Fanuc TP program (LS listing): S005.LS

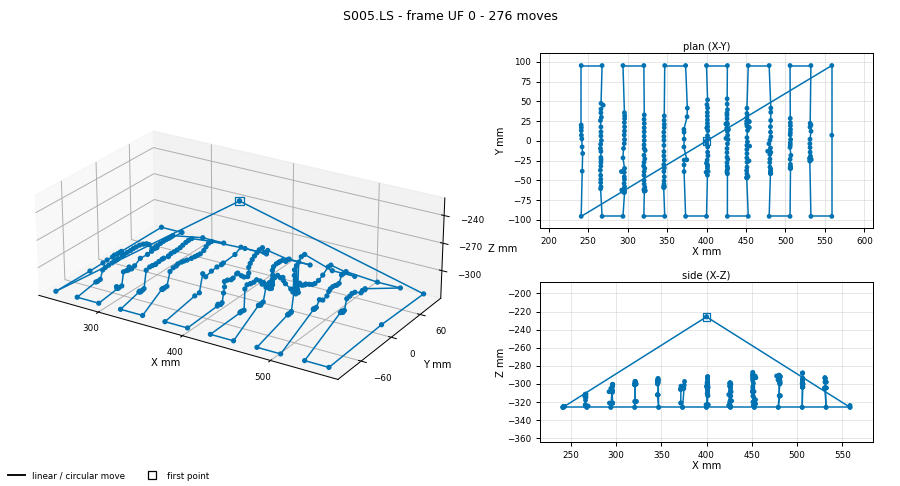
[picture p0: tool path of S005.LS in frame UF 0, 276 of 276 moves have a stored position in this frame; points joined in program order, loops and branches not executed]
/PROG  S005.LS
/ATTR
OWNER       = MNEDITOR;
COMMENT     = "";
PROG_SIZE   = 636;
CREATE      = DATE 23-01-07  TIME 11:59:14;
MODIFIED    = DATE 23-01-07  TIME 12:02:18;
FILE_NAME   = ;
VERSION     = 0;
LINE_COUNT  = 4;
MEMORY_SIZE = 992;
PROTECT     = READ_WRITE;
TCD:  STACK_SIZE    = 0,
      TASK_PRIORITY = 50,
      TIME_SLICE    = 0,
      BUSY_LAMP_OFF = 0,
      ABORT_REQUEST = 0,
      PAUSE_REQUEST = 0;
DEFAULT_GROUP    = 1,*,*,*,*;
CONTROL_CODE     = 00000000 00000000;
/MN
   1:J P[1] 100% FINE    ;
   2:L P[2] 300mm/sec CNT100    ;
   3:L P[3] 300mm/sec CNT100    ;
   4:L P[4] 300mm/sec CNT100    ;
   5:L P[5] 300mm/sec CNT100    ;
   6:L P[6] 300mm/sec CNT100    ;
   7:L P[7] 300mm/sec CNT100    ;
   8:L P[8] 300mm/sec CNT100    ;
   9:L P[9] 300mm/sec CNT100    ;
   10:L P[10] 300mm/sec CNT100    ;
   11:L P[11] 300mm/sec CNT100    ;
   12:L P[12] 300mm/sec CNT100    ;
   13:L P[13] 300mm/sec CNT100    ;
   14:L P[14] 300mm/sec CNT100    ;
   15:L P[15] 300mm/sec CNT100    ;
   16:L P[16] 300mm/sec CNT100    ;
   17:L P[17] 300mm/sec CNT100    ;
   18:L P[18] 300mm/sec CNT100    ;
   19:L P[19] 300mm/sec CNT100    ;
   20:L P[20] 300mm/sec CNT100    ;
   21:L P[21] 300mm/sec CNT100    ;
   22:L P[22] 300mm/sec CNT100    ;
   23:L P[23] 300mm/sec CNT100    ;
   24:L P[24] 300mm/sec CNT100    ;
   25:L P[25] 300mm/sec CNT100    ;
   26:L P[26] 300mm/sec CNT100    ;
   27:L P[27] 300mm/sec CNT100    ;
   28:L P[28] 300mm/sec CNT100    ;
   29:L P[29] 300mm/sec CNT100    ;
   30:L P[30] 300mm/sec CNT100    ;
   31:L P[31] 300mm/sec CNT100    ;
   32:L P[32] 300mm/sec CNT100    ;
   33:L P[33] 300mm/sec CNT100    ;
   34:L P[34] 300mm/sec CNT100    ;
   35:L P[35] 300mm/sec CNT100    ;
   36:L P[36] 300mm/sec CNT100    ;
   37:L P[37] 300mm/sec CNT100    ;
   38:L P[38] 300mm/sec CNT100    ;
   39:L P[39] 300mm/sec CNT100    ;
   40:L P[40] 300mm/sec CNT100    ;
   41:L P[41] 300mm/sec CNT100    ;
   42:L P[42] 300mm/sec CNT100    ;
   43:L P[43] 300mm/sec CNT100    ;
   44:L P[44] 300mm/sec CNT100    ;
   45:L P[45] 300mm/sec CNT100    ;
   46:L P[46] 300mm/sec CNT100    ;
   47:L P[47] 300mm/sec CNT100    ;
   48:L P[48] 300mm/sec CNT100    ;
   49:L P[49] 300mm/sec CNT100    ;
   50:L P[50] 300mm/sec CNT100    ;
   51:L P[51] 300mm/sec CNT100    ;
   52:L P[52] 300mm/sec CNT100    ;
   53:L P[53] 300mm/sec CNT100    ;
   54:L P[54] 300mm/sec CNT100    ;
   55:L P[55] 300mm/sec CNT100    ;
   56:L P[56] 300mm/sec CNT100    ;
   57:L P[57] 300mm/sec CNT100    ;
   58:L P[58] 300mm/sec CNT100    ;
   59:L P[59] 300mm/sec CNT100    ;
   60:L P[60] 300mm/sec CNT100    ;
   61:L P[61] 300mm/sec CNT100    ;
   62:L P[62] 300mm/sec CNT100    ;
   63:L P[63] 300mm/sec CNT100    ;
   64:L P[64] 300mm/sec CNT100    ;
   65:L P[65] 300mm/sec CNT100    ;
   66:L P[66] 300mm/sec CNT100    ;
   67:L P[67] 300mm/sec CNT100    ;
   68:L P[68] 300mm/sec CNT100    ;
   69:L P[69] 300mm/sec CNT100    ;
   70:L P[70] 300mm/sec CNT100    ;
   71:L P[71] 300mm/sec CNT100    ;
   72:L P[72] 300mm/sec CNT100    ;
   73:L P[73] 300mm/sec CNT100    ;
   74:L P[74] 300mm/sec CNT100    ;
   75:L P[75] 300mm/sec CNT100    ;
   76:L P[76] 300mm/sec CNT100    ;
   77:L P[77] 300mm/sec CNT100    ;
   78:L P[78] 300mm/sec CNT100    ;
   79:L P[79] 300mm/sec CNT100    ;
   80:L P[80] 300mm/sec CNT100    ;
   81:L P[81] 300mm/sec CNT100    ;
   82:L P[82] 300mm/sec CNT100    ;
   83:L P[83] 300mm/sec CNT100    ;
   84:L P[84] 300mm/sec CNT100    ;
   85:L P[85] 300mm/sec CNT100    ;
   86:L P[86] 300mm/sec CNT100    ;
   87:L P[87] 300mm/sec CNT100    ;
   88:L P[88] 300mm/sec CNT100    ;
   89:L P[89] 300mm/sec CNT100    ;
   90:L P[90] 300mm/sec CNT100    ;
   91:L P[91] 300mm/sec CNT100    ;
   92:L P[92] 300mm/sec CNT100    ;
   93:L P[93] 300mm/sec CNT100    ;
   94:L P[94] 300mm/sec CNT100    ;
   95:L P[95] 300mm/sec CNT100    ;
   96:L P[96] 300mm/sec CNT100    ;
   97:L P[97] 300mm/sec CNT100    ;
   98:L P[98] 300mm/sec CNT100    ;
   99:L P[99] 300mm/sec CNT100    ;
   100:L P[100] 300mm/sec CNT100    ;
   101:L P[101] 300mm/sec CNT100    ;
   102:L P[102] 300mm/sec CNT100    ;
   103:L P[103] 300mm/sec CNT100    ;
   104:L P[104] 300mm/sec CNT100    ;
   105:L P[105] 300mm/sec CNT100    ;
   106:L P[106] 300mm/sec CNT100    ;
   107:L P[107] 300mm/sec CNT100    ;
   108:L P[108] 300mm/sec CNT100    ;
   109:L P[109] 300mm/sec CNT100    ;
   110:L P[110] 300mm/sec CNT100    ;
   111:L P[111] 300mm/sec CNT100    ;
   112:L P[112] 300mm/sec CNT100    ;
   113:L P[113] 300mm/sec CNT100    ;
   114:L P[114] 300mm/sec CNT100    ;
   115:L P[115] 300mm/sec CNT100    ;
   116:L P[116] 300mm/sec CNT100    ;
   117:L P[117] 300mm/sec CNT100    ;
   118:L P[118] 300mm/sec CNT100    ;
   119:L P[119] 300mm/sec CNT100    ;
   120:L P[120] 300mm/sec CNT100    ;
   121:L P[121] 300mm/sec CNT100    ;
   122:L P[122] 300mm/sec CNT100    ;
   123:L P[123] 300mm/sec CNT100    ;
   124:L P[124] 300mm/sec CNT100    ;
   125:L P[125] 300mm/sec CNT100    ;
   126:L P[126] 300mm/sec CNT100    ;
   127:L P[127] 300mm/sec CNT100    ;
   128:L P[128] 300mm/sec CNT100    ;
   129:L P[129] 300mm/sec CNT100    ;
   130:L P[130] 300mm/sec CNT100    ;
   131:L P[131] 300mm/sec CNT100    ;
   132:L P[132] 300mm/sec CNT100    ;
   133:L P[133] 300mm/sec CNT100    ;
   134:L P[134] 300mm/sec CNT100    ;
   135:L P[135] 300mm/sec CNT100    ;
   136:L P[136] 300mm/sec CNT100    ;
   137:L P[137] 300mm/sec CNT100    ;
   138:L P[138] 300mm/sec CNT100    ;
   139:L P[139] 300mm/sec CNT100    ;
   140:L P[140] 300mm/sec CNT100    ;
   141:L P[141] 300mm/sec CNT100    ;
   142:L P[142] 300mm/sec CNT100    ;
   143:L P[143] 300mm/sec CNT100    ;
   144:L P[144] 300mm/sec CNT100    ;
   145:L P[145] 300mm/sec CNT100    ;
   146:L P[146] 300mm/sec CNT100    ;
   147:L P[147] 300mm/sec CNT100    ;
   148:L P[148] 300mm/sec CNT100    ;
   149:L P[149] 300mm/sec CNT100    ;
   150:L P[150] 300mm/sec CNT100    ;
   151:L P[151] 300mm/sec CNT100    ;
   152:L P[152] 300mm/sec CNT100    ;
   153:L P[153] 300mm/sec CNT100    ;
   154:L P[154] 300mm/sec CNT100    ;
   155:L P[155] 300mm/sec CNT100    ;
   156:L P[156] 300mm/sec CNT100    ;
   157:L P[157] 300mm/sec CNT100    ;
   158:L P[158] 300mm/sec CNT100    ;
   159:L P[159] 300mm/sec CNT100    ;
   160:L P[160] 300mm/sec CNT100    ;
   161:L P[161] 300mm/sec CNT100    ;
   162:L P[162] 300mm/sec CNT100    ;
   163:L P[163] 300mm/sec CNT100    ;
   164:L P[164] 300mm/sec CNT100    ;
   165:L P[165] 300mm/sec CNT100    ;
   166:L P[166] 300mm/sec CNT100    ;
   167:L P[167] 300mm/sec CNT100    ;
   168:L P[168] 300mm/sec CNT100    ;
   169:L P[169] 300mm/sec CNT100    ;
   170:L P[170] 300mm/sec CNT100    ;
   171:L P[171] 300mm/sec CNT100    ;
   172:L P[172] 300mm/sec CNT100    ;
   173:L P[173] 300mm/sec CNT100    ;
   174:L P[174] 300mm/sec CNT100    ;
   175:L P[175] 300mm/sec CNT100    ;
   176:L P[176] 300mm/sec CNT100    ;
   177:L P[177] 300mm/sec CNT100    ;
   178:L P[178] 300mm/sec CNT100    ;
   179:L P[179] 300mm/sec CNT100    ;
   180:L P[180] 300mm/sec CNT100    ;
   181:L P[181] 300mm/sec CNT100    ;
   182:L P[182] 300mm/sec CNT100    ;
   183:L P[183] 300mm/sec CNT100    ;
   184:L P[184] 300mm/sec CNT100    ;
   185:L P[185] 300mm/sec CNT100    ;
   186:L P[186] 300mm/sec CNT100    ;
   187:L P[187] 300mm/sec CNT100    ;
   188:L P[188] 300mm/sec CNT100    ;
   189:L P[189] 300mm/sec CNT100    ;
   190:L P[190] 300mm/sec CNT100    ;
   191:L P[191] 300mm/sec CNT100    ;
   192:L P[192] 300mm/sec CNT100    ;
   193:L P[193] 300mm/sec CNT100    ;
   194:L P[194] 300mm/sec CNT100    ;
   195:L P[195] 300mm/sec CNT100    ;
   196:L P[196] 300mm/sec CNT100    ;
   197:L P[197] 300mm/sec CNT100    ;
   198:L P[198] 300mm/sec CNT100    ;
   199:L P[199] 300mm/sec CNT100    ;
   200:L P[200] 300mm/sec CNT100    ;
   201:L P[201] 300mm/sec CNT100    ;
   202:L P[202] 300mm/sec CNT100    ;
   203:L P[203] 300mm/sec CNT100    ;
   204:L P[204] 300mm/sec CNT100    ;
   205:L P[205] 300mm/sec CNT100    ;
   206:L P[206] 300mm/sec CNT100    ;
   207:L P[207] 300mm/sec CNT100    ;
   208:L P[208] 300mm/sec CNT100    ;
   209:L P[209] 300mm/sec CNT100    ;
   210:L P[210] 300mm/sec CNT100    ;
   211:L P[211] 300mm/sec CNT100    ;
   212:L P[212] 300mm/sec CNT100    ;
   213:L P[213] 300mm/sec CNT100    ;
   214:L P[214] 300mm/sec CNT100    ;
   215:L P[215] 300mm/sec CNT100    ;
   216:L P[216] 300mm/sec CNT100    ;
   217:L P[217] 300mm/sec CNT100    ;
   218:L P[218] 300mm/sec CNT100    ;
   219:L P[219] 300mm/sec CNT100    ;
   220:L P[220] 300mm/sec CNT100    ;
   221:L P[221] 300mm/sec CNT100    ;
   222:L P[222] 300mm/sec CNT100    ;
   223:L P[223] 300mm/sec CNT100    ;
   224:L P[224] 300mm/sec CNT100    ;
   225:L P[225] 300mm/sec CNT100    ;
   226:L P[226] 300mm/sec CNT100    ;
   227:L P[227] 300mm/sec CNT100    ;
   228:L P[228] 300mm/sec CNT100    ;
   229:L P[229] 300mm/sec CNT100    ;
   230:L P[230] 300mm/sec CNT100    ;
   231:L P[231] 300mm/sec CNT100    ;
   232:L P[232] 300mm/sec CNT100    ;
   233:L P[233] 300mm/sec CNT100    ;
   234:L P[234] 300mm/sec CNT100    ;
   235:L P[235] 300mm/sec CNT100    ;
   236:L P[236] 300mm/sec CNT100    ;
   237:L P[237] 300mm/sec CNT100    ;
   238:L P[238] 300mm/sec CNT100    ;
   239:L P[239] 300mm/sec CNT100    ;
   240:L P[240] 300mm/sec CNT100    ;
   241:L P[241] 300mm/sec CNT100    ;
   242:L P[242] 300mm/sec CNT100    ;
   243:L P[243] 300mm/sec CNT100    ;
   244:L P[244] 300mm/sec CNT100    ;
   245:L P[245] 300mm/sec CNT100    ;
   246:L P[246] 300mm/sec CNT100    ;
   247:L P[247] 300mm/sec CNT100    ;
   248:L P[248] 300mm/sec CNT100    ;
   249:L P[249] 300mm/sec CNT100    ;
   250:L P[250] 300mm/sec CNT100    ;
   251:L P[251] 300mm/sec CNT100    ;
   252:L P[252] 300mm/sec CNT100    ;
   253:L P[253] 300mm/sec CNT100    ;
   254:L P[254] 300mm/sec CNT100    ;
   255:L P[255] 300mm/sec CNT100    ;
   256:L P[256] 300mm/sec CNT100    ;
   257:L P[257] 300mm/sec CNT100    ;
   258:L P[258] 300mm/sec CNT100    ;
   259:L P[259] 300mm/sec CNT100    ;
   260:L P[260] 300mm/sec CNT100    ;
   261:L P[261] 300mm/sec CNT100    ;
   262:L P[262] 300mm/sec CNT100    ;
   263:L P[263] 300mm/sec CNT100    ;
   264:L P[264] 300mm/sec CNT100    ;
   265:L P[265] 300mm/sec CNT100    ;
   266:L P[266] 300mm/sec CNT100    ;
   267:L P[267] 300mm/sec CNT100    ;
   268:L P[268] 300mm/sec CNT100    ;
   269:L P[269] 300mm/sec CNT100    ;
   270:L P[270] 300mm/sec CNT100    ;
   271:L P[271] 300mm/sec CNT100    ;
   272:L P[272] 300mm/sec CNT100    ;
   273:L P[273] 300mm/sec CNT100    ;
   274:L P[274] 300mm/sec CNT100    ;
   275:L P[275] 300mm/sec CNT100    ;
   276:L P[276] 300mm/sec CNT100    ;
/POS
P[1]{
   GP1:
    UF : 0, UT : 6,      CONFIG : 'N U T, 0, 0, 0',
    X =  400.000  mm,    Y =   0.000  mm,    Z =   -225.827  mm,
    W =  -180.000 deg,    P =   0.000 deg,    R =   0.000 deg
};
P[2]{
   GP1:
    UF : 0, UT : 6,      CONFIG : 'N U T, 0, 0, 0',
    X =  558.634  mm,    Y =   95.475  mm,    Z =   -325.827  mm,
    W =  -180.000 deg,    P =   0.000 deg,    R =   0.000 deg
};
P[3]{
   GP1:
    UF : 0, UT : 6,      CONFIG : 'N U T, 0, 0, 0',
    X =  558.634  mm,    Y =   7.217  mm,    Z =   -323.775  mm,
    W =  -191.515 deg,    P =   0.198 deg,    R =   -0.974 deg
};
P[4]{
   GP1:
    UF : 0, UT : 6,      CONFIG : 'N U T, 0, 0, 0',
    X =  558.634  mm,    Y =   -95.475  mm,    Z =   -325.827  mm,
    W =  -180.000 deg,    P =   0.000 deg,    R =   0.000 deg
};
P[5]{
   GP1:
    UF : 0, UT : 6,      CONFIG : 'N U T, 0, 0, 0',
    X =  532.195  mm,    Y =   -95.475  mm,    Z =   -325.827  mm,
    W =  -180.000 deg,    P =   0.000 deg,    R =   0.000 deg
};
P[6]{
   GP1:
    UF : 0, UT : 6,      CONFIG : 'N U T, 0, 0, 0',
    X =  530.814  mm,    Y =   -25.583  mm,    Z =   -304.407  mm,
    W =  -188.861 deg,    P =   0.154 deg,    R =   -0.988 deg
};
P[7]{
   GP1:
    UF : 0, UT : 6,      CONFIG : 'N U T, 0, 0, 0',
    X =  530.964  mm,    Y =   -24.537  mm,    Z =   -304.407  mm,
    W =  -188.880 deg,    P =   0.154 deg,    R =   -0.988 deg
};
P[8]{
   GP1:
    UF : 0, UT : 6,      CONFIG : 'N U T, 0, 0, 0',
    X =  532.628  mm,    Y =   -23.681  mm,    Z =   -304.407  mm,
    W =  -189.388 deg,    P =   0.163 deg,    R =   -0.986 deg
};
P[9]{
   GP1:
    UF : 0, UT : 6,      CONFIG : 'N U T, 0, 0, 0',
    X =  531.884  mm,    Y =   -22.450  mm,    Z =   -304.407  mm,
    W =  -188.725 deg,    P =   0.152 deg,    R =   -0.988 deg
};
P[10]{
   GP1:
    UF : 0, UT : 6,      CONFIG : 'N U T, 0, 0, 0',
    X =  530.384  mm,    Y =   -21.896  mm,    Z =   -304.407  mm,
    W =  -188.440 deg,    P =   0.147 deg,    R =   -0.989 deg
};
P[11]{
   GP1:
    UF : 0, UT : 6,      CONFIG : 'N U T, 0, 0, 0',
    X =  531.596  mm,    Y =   -19.218  mm,    Z =   -304.407  mm,
    W =  -188.563 deg,    P =   0.149 deg,    R =   -0.989 deg
};
P[12]{
   GP1:
    UF : 0, UT : 6,      CONFIG : 'N U T, 0, 0, 0',
    X =  531.190  mm,    Y =   -14.198  mm,    Z =   -294.050  mm,
    W =  -188.299 deg,    P =   0.144 deg,    R =   -0.989 deg
};
P[13]{
   GP1:
    UF : 0, UT : 6,      CONFIG : 'N U T, 0, 0, 0',
    X =  531.084  mm,    Y =   -8.401  mm,    Z =   -293.746  mm,
    W =  -188.006 deg,    P =   0.139 deg,    R =   -0.990 deg
};
P[14]{
   GP1:
    UF : 0, UT : 6,      CONFIG : 'N U T, 0, 0, 0',
    X =  530.854  mm,    Y =   -3.421  mm,    Z =   -292.906  mm,
    W =  -187.902 deg,    P =   0.137 deg,    R =   -0.990 deg
};
P[15]{
   GP1:
    UF : 0, UT : 6,      CONFIG : 'N U T, 0, 0, 0',
    X =  531.042  mm,    Y =   2.169  mm,    Z =   -293.703  mm,
    W =  -187.687 deg,    P =   0.134 deg,    R =   -0.991 deg
};
P[16]{
   GP1:
    UF : 0, UT : 6,      CONFIG : 'N U T, 0, 0, 0',
    X =  532.332  mm,    Y =   12.263  mm,    Z =   -297.988  mm,
    W =  -187.056 deg,    P =   0.123 deg,    R =   -0.992 deg
};
P[17]{
   GP1:
    UF : 0, UT : 6,      CONFIG : 'N U T, 0, 0, 0',
    X =  531.017  mm,    Y =   17.469  mm,    Z =   -297.873  mm,
    W =  -186.987 deg,    P =   0.122 deg,    R =   -0.992 deg
};
P[18]{
   GP1:
    UF : 0, UT : 6,      CONFIG : 'N U T, 0, 0, 0',
    X =  532.240  mm,    Y =   20.203  mm,    Z =   -297.873  mm,
    W =  -186.760 deg,    P =   0.118 deg,    R =   -0.993 deg
};
P[19]{
   GP1:
    UF : 0, UT : 6,      CONFIG : 'N U T, 0, 0, 0',
    X =  531.259  mm,    Y =   22.383  mm,    Z =   -297.873  mm,
    W =  -186.691 deg,    P =   0.116 deg,    R =   -0.993 deg
};
P[20]{
   GP1:
    UF : 0, UT : 6,      CONFIG : 'N U T, 0, 0, 0',
    X =  532.195  mm,    Y =   95.475  mm,    Z =   -325.827  mm,
    W =  -180.000 deg,    P =   0.000 deg,    R =   0.000 deg
};
P[21]{
   GP1:
    UF : 0, UT : 6,      CONFIG : 'N U T, 0, 0, 0',
    X =  505.756  mm,    Y =   95.475  mm,    Z =   -325.827  mm,
    W =  -180.000 deg,    P =   0.000 deg,    R =   0.000 deg
};
P[22]{
   GP1:
    UF : 0, UT : 6,      CONFIG : 'N U T, 0, 0, 0',
    X =  506.048  mm,    Y =   28.588  mm,    Z =   -287.949  mm,
    W =  -185.682 deg,    P =   0.099 deg,    R =   -0.995 deg
};
P[23]{
   GP1:
    UF : 0, UT : 6,      CONFIG : 'N U T, 0, 0, 0',
    X =  506.139  mm,    Y =   23.053  mm,    Z =   -287.949  mm,
    W =  -186.283 deg,    P =   0.109 deg,    R =   -0.993 deg
};
P[24]{
   GP1:
    UF : 0, UT : 6,      CONFIG : 'N U T, 0, 0, 0',
    X =  506.242  mm,    Y =   19.243  mm,    Z =   -287.949  mm,
    W =  -186.576 deg,    P =   0.114 deg,    R =   -0.993 deg
};
P[25]{
   GP1:
    UF : 0, UT : 6,      CONFIG : 'N U T, 0, 0, 0',
    X =  506.313  mm,    Y =   14.626  mm,    Z =   -295.171  mm,
    W =  -186.784 deg,    P =   0.118 deg,    R =   -0.992 deg
};
P[26]{
   GP1:
    UF : 0, UT : 6,      CONFIG : 'N U T, 0, 0, 0',
    X =  506.148  mm,    Y =   10.652  mm,    Z =   -295.522  mm,
    W =  -186.971 deg,    P =   0.121 deg,    R =   -0.992 deg
};
P[27]{
   GP1:
    UF : 0, UT : 6,      CONFIG : 'N U T, 0, 0, 0',
    X =  505.935  mm,    Y =   7.694  mm,    Z =   -294.830  mm,
    W =  -187.017 deg,    P =   0.122 deg,    R =   -0.992 deg
};
P[28]{
   GP1:
    UF : 0, UT : 6,      CONFIG : 'N U T, 0, 0, 0',
    X =  506.494  mm,    Y =   1.825  mm,    Z =   -293.624  mm,
    W =  -187.247 deg,    P =   0.126 deg,    R =   -0.991 deg
};
P[29]{
   GP1:
    UF : 0, UT : 6,      CONFIG : 'N U T, 0, 0, 0',
    X =  506.090  mm,    Y =   -2.448  mm,    Z =   -294.465  mm,
    W =  -187.355 deg,    P =   0.128 deg,    R =   -0.991 deg
};
P[30]{
   GP1:
    UF : 0, UT : 6,      CONFIG : 'N U T, 0, 0, 0',
    X =  506.095  mm,    Y =   -5.498  mm,    Z =   -296.134  mm,
    W =  -187.464 deg,    P =   0.130 deg,    R =   -0.991 deg
};
P[31]{
   GP1:
    UF : 0, UT : 6,      CONFIG : 'N U T, 0, 0, 0',
    X =  505.684  mm,    Y =   -8.195  mm,    Z =   -299.862  mm,
    W =  -187.766 deg,    P =   0.135 deg,    R =   -0.990 deg
};
P[32]{
   GP1:
    UF : 0, UT : 6,      CONFIG : 'N U T, 0, 0, 0',
    X =  506.835  mm,    Y =   -18.194  mm,    Z =   -300.042  mm,
    W =  -188.013 deg,    P =   0.139 deg,    R =   -0.990 deg
};
P[33]{
   GP1:
    UF : 0, UT : 6,      CONFIG : 'N U T, 0, 0, 0',
    X =  505.884  mm,    Y =   -23.144  mm,    Z =   -297.872  mm,
    W =  -188.330 deg,    P =   0.145 deg,    R =   -0.989 deg
};
P[34]{
   GP1:
    UF : 0, UT : 6,      CONFIG : 'N U T, 0, 0, 0',
    X =  506.212  mm,    Y =   -29.601  mm,    Z =   -303.408  mm,
    W =  -188.657 deg,    P =   0.150 deg,    R =   -0.988 deg
};
P[35]{
   GP1:
    UF : 0, UT : 6,      CONFIG : 'N U T, 0, 0, 0',
    X =  506.536  mm,    Y =   -32.853  mm,    Z =   -303.408  mm,
    W =  -188.193 deg,    P =   0.142 deg,    R =   -0.989 deg
};
P[36]{
   GP1:
    UF : 0, UT : 6,      CONFIG : 'N U T, 0, 0, 0',
    X =  506.007  mm,    Y =   -33.420  mm,    Z =   -303.408  mm,
    W =  -188.300 deg,    P =   0.144 deg,    R =   -0.989 deg
};
P[37]{
   GP1:
    UF : 0, UT : 6,      CONFIG : 'N U T, 0, 0, 0',
    X =  506.223  mm,    Y =   -33.762  mm,    Z =   -303.408  mm,
    W =  -188.800 deg,    P =   0.153 deg,    R =   -0.988 deg
};
P[38]{
   GP1:
    UF : 0, UT : 6,      CONFIG : 'N U T, 0, 0, 0',
    X =  506.351  mm,    Y =   -34.485  mm,    Z =   -303.408  mm,
    W =  -188.415 deg,    P =   0.146 deg,    R =   -0.989 deg
};
P[39]{
   GP1:
    UF : 0, UT : 6,      CONFIG : 'N U T, 0, 0, 0',
    X =  505.879  mm,    Y =   -34.702  mm,    Z =   -303.408  mm,
    W =  -188.522 deg,    P =   0.148 deg,    R =   -0.988 deg
};
P[40]{
   GP1:
    UF : 0, UT : 6,      CONFIG : 'N U T, 0, 0, 0',
    X =  506.333  mm,    Y =   -34.799  mm,    Z =   -303.408  mm,
    W =  -188.722 deg,    P =   0.152 deg,    R =   -0.988 deg
};
P[41]{
   GP1:
    UF : 0, UT : 6,      CONFIG : 'N U T, 0, 0, 0',
    X =  505.756  mm,    Y =   -95.475  mm,    Z =   -325.827  mm,
    W =  -180.000 deg,    P =   0.000 deg,    R =   0.000 deg
};
P[42]{
   GP1:
    UF : 0, UT : 6,      CONFIG : 'N U T, 0, 0, 0',
    X =  479.317  mm,    Y =   -95.475  mm,    Z =   -325.827  mm,
    W =  -180.000 deg,    P =   0.000 deg,    R =   0.000 deg
};
P[43]{
   GP1:
    UF : 0, UT : 6,      CONFIG : 'N U T, 0, 0, 0',
    X =  480.938  mm,    Y =   -41.376  mm,    Z =   -313.087  mm,
    W =  -188.017 deg,    P =   0.139 deg,    R =   -0.989 deg
};
P[44]{
   GP1:
    UF : 0, UT : 6,      CONFIG : 'N U T, 0, 0, 0',
    X =  481.407  mm,    Y =   -41.075  mm,    Z =   -313.087  mm,
    W =  -188.113 deg,    P =   0.141 deg,    R =   -0.988 deg
};
P[45]{
   GP1:
    UF : 0, UT : 6,      CONFIG : 'N U T, 0, 0, 0',
    X =  481.271  mm,    Y =   -40.084  mm,    Z =   -313.087  mm,
    W =  -188.018 deg,    P =   0.139 deg,    R =   -0.989 deg
};
P[46]{
   GP1:
    UF : 0, UT : 6,      CONFIG : 'N U T, 0, 0, 0',
    X =  481.091  mm,    Y =   -38.858  mm,    Z =   -313.087  mm,
    W =  -188.196 deg,    P =   0.142 deg,    R =   -0.988 deg
};
P[47]{
   GP1:
    UF : 0, UT : 6,      CONFIG : 'N U T, 0, 0, 0',
    X =  480.891  mm,    Y =   -38.855  mm,    Z =   -313.087  mm,
    W =  -188.007 deg,    P =   0.139 deg,    R =   -0.989 deg
};
P[48]{
   GP1:
    UF : 0, UT : 6,      CONFIG : 'N U T, 0, 0, 0',
    X =  481.242  mm,    Y =   -35.551  mm,    Z =   -313.087  mm,
    W =  -188.243 deg,    P =   0.143 deg,    R =   -0.988 deg
};
P[49]{
   GP1:
    UF : 0, UT : 6,      CONFIG : 'N U T, 0, 0, 0',
    X =  480.348  mm,    Y =   -33.106  mm,    Z =   -313.087  mm,
    W =  -188.280 deg,    P =   0.144 deg,    R =   -0.988 deg
};
P[50]{
   GP1:
    UF : 0, UT : 6,      CONFIG : 'N U T, 0, 0, 0',
    X =  480.001  mm,    Y =   -27.363  mm,    Z =   -290.743  mm,
    W =  -188.245 deg,    P =   0.143 deg,    R =   -0.988 deg
};
P[51]{
   GP1:
    UF : 0, UT : 6,      CONFIG : 'N U T, 0, 0, 0',
    X =  480.299  mm,    Y =   -22.934  mm,    Z =   -290.231  mm,
    W =  -188.240 deg,    P =   0.143 deg,    R =   -0.988 deg
};
P[52]{
   GP1:
    UF : 0, UT : 6,      CONFIG : 'N U T, 0, 0, 0',
    X =  480.195  mm,    Y =   -17.131  mm,    Z =   -290.663  mm,
    W =  -188.197 deg,    P =   0.142 deg,    R =   -0.988 deg
};
P[53]{
   GP1:
    UF : 0, UT : 6,      CONFIG : 'N U T, 0, 0, 0',
    X =  481.449  mm,    Y =   -14.408  mm,    Z =   -291.912  mm,
    W =  -188.071 deg,    P =   0.140 deg,    R =   -0.989 deg
};
P[54]{
   GP1:
    UF : 0, UT : 6,      CONFIG : 'N U T, 0, 0, 0',
    X =  477.486  mm,    Y =   -12.964  mm,    Z =   -291.185  mm,
    W =  -188.218 deg,    P =   0.143 deg,    R =   -0.988 deg
};
P[55]{
   GP1:
    UF : 0, UT : 6,      CONFIG : 'N U T, 0, 0, 0',
    X =  480.965  mm,    Y =   -8.815  mm,    Z =   -293.764  mm,
    W =  -188.087 deg,    P =   0.140 deg,    R =   -0.989 deg
};
P[56]{
   GP1:
    UF : 0, UT : 6,      CONFIG : 'N U T, 0, 0, 0',
    X =  478.982  mm,    Y =   -3.456  mm,    Z =   -295.473  mm,
    W =  -188.273 deg,    P =   0.144 deg,    R =   -0.988 deg
};
P[57]{
   GP1:
    UF : 0, UT : 6,      CONFIG : 'N U T, 0, 0, 0',
    X =  480.338  mm,    Y =   1.052  mm,    Z =   -297.298  mm,
    W =  -188.237 deg,    P =   0.143 deg,    R =   -0.988 deg
};
P[58]{
   GP1:
    UF : 0, UT : 6,      CONFIG : 'N U T, 0, 0, 0',
    X =  481.501  mm,    Y =   5.284  mm,    Z =   -298.867  mm,
    W =  -188.194 deg,    P =   0.142 deg,    R =   -0.988 deg
};
P[59]{
   GP1:
    UF : 0, UT : 6,      CONFIG : 'N U T, 0, 0, 0',
    X =  481.028  mm,    Y =   11.149  mm,    Z =   -300.166  mm,
    W =  -188.241 deg,    P =   0.143 deg,    R =   -0.988 deg
};
P[60]{
   GP1:
    UF : 0, UT : 6,      CONFIG : 'N U T, 0, 0, 0',
    X =  480.986  mm,    Y =   18.030  mm,    Z =   -299.581  mm,
    W =  -188.105 deg,    P =   0.141 deg,    R =   -0.989 deg
};
P[61]{
   GP1:
    UF : 0, UT : 6,      CONFIG : 'N U T, 0, 0, 0',
    X =  481.262  mm,    Y =   25.935  mm,    Z =   -296.771  mm,
    W =  -187.857 deg,    P =   0.137 deg,    R =   -0.989 deg
};
P[62]{
   GP1:
    UF : 0, UT : 6,      CONFIG : 'N U T, 0, 0, 0',
    X =  481.355  mm,    Y =   36.326  mm,    Z =   -291.876  mm,
    W =  -187.261 deg,    P =   0.126 deg,    R =   -0.991 deg
};
P[63]{
   GP1:
    UF : 0, UT : 6,      CONFIG : 'N U T, 0, 0, 0',
    X =  481.444  mm,    Y =   41.651  mm,    Z =   -291.876  mm,
    W =  -186.873 deg,    P =   0.120 deg,    R =   -0.992 deg
};
P[64]{
   GP1:
    UF : 0, UT : 6,      CONFIG : 'N U T, 0, 0, 0',
    X =  479.317  mm,    Y =   95.475  mm,    Z =   -325.827  mm,
    W =  -180.000 deg,    P =   0.000 deg,    R =   0.000 deg
};
P[65]{
   GP1:
    UF : 0, UT : 6,      CONFIG : 'N U T, 0, 0, 0',
    X =  452.878  mm,    Y =   95.475  mm,    Z =   -325.827  mm,
    W =  -180.000 deg,    P =   0.000 deg,    R =   0.000 deg
};
P[66]{
   GP1:
    UF : 0, UT : 6,      CONFIG : 'N U T, 0, 0, 0',
    X =  451.197  mm,    Y =   41.411  mm,    Z =   -287.331  mm,
    W =  -187.870 deg,    P =   0.137 deg,    R =   -0.988 deg
};
P[67]{
   GP1:
    UF : 0, UT : 6,      CONFIG : 'N U T, 0, 0, 0',
    X =  451.191  mm,    Y =   34.711  mm,    Z =   -287.331  mm,
    W =  -188.504 deg,    P =   0.148 deg,    R =   -0.987 deg
};
P[68]{
   GP1:
    UF : 0, UT : 6,      CONFIG : 'N U T, 0, 0, 0',
    X =  451.188  mm,    Y =   29.919  mm,    Z =   -291.318  mm,
    W =  -188.638 deg,    P =   0.150 deg,    R =   -0.987 deg
};
P[69]{
   GP1:
    UF : 0, UT : 6,      CONFIG : 'N U T, 0, 0, 0',
    X =  452.779  mm,    Y =   25.537  mm,    Z =   -319.697  mm,
    W =  -188.810 deg,    P =   0.153 deg,    R =   -0.987 deg
};
P[70]{
   GP1:
    UF : 0, UT : 6,      CONFIG : 'N U T, 0, 0, 0',
    X =  451.187  mm,    Y =   25.392  mm,    Z =   -293.474  mm,
    W =  -188.698 deg,    P =   0.151 deg,    R =   -0.987 deg
};
P[71]{
   GP1:
    UF : 0, UT : 6,      CONFIG : 'N U T, 0, 0, 0',
    X =  451.265  mm,    Y =   24.845  mm,    Z =   -313.269  mm,
    W =  -188.891 deg,    P =   0.154 deg,    R =   -0.986 deg
};
P[72]{
   GP1:
    UF : 0, UT : 6,      CONFIG : 'N U T, 0, 0, 0',
    X =  454.277  mm,    Y =   24.387  mm,    Z =   -322.007  mm,
    W =  -188.827 deg,    P =   0.153 deg,    R =   -0.986 deg
};
P[73]{
   GP1:
    UF : 0, UT : 6,      CONFIG : 'N U T, 0, 0, 0',
    X =  451.681  mm,    Y =   23.888  mm,    Z =   -323.972  mm,
    W =  -188.865 deg,    P =   0.154 deg,    R =   -0.986 deg
};
P[74]{
   GP1:
    UF : 0, UT : 6,      CONFIG : 'N U T, 0, 0, 0',
    X =  451.241  mm,    Y =   23.186  mm,    Z =   -308.112  mm,
    W =  -188.788 deg,    P =   0.153 deg,    R =   -0.987 deg
};
P[75]{
   GP1:
    UF : 0, UT : 6,      CONFIG : 'N U T, 0, 0, 0',
    X =  451.191  mm,    Y =   21.539  mm,    Z =   -296.623  mm,
    W =  -188.766 deg,    P =   0.152 deg,    R =   -0.987 deg
};
P[76]{
   GP1:
    UF : 0, UT : 6,      CONFIG : 'N U T, 0, 0, 0',
    X =  451.216  mm,    Y =   21.316  mm,    Z =   -302.688  mm,
    W =  -188.807 deg,    P =   0.153 deg,    R =   -0.987 deg
};
P[77]{
   GP1:
    UF : 0, UT : 6,      CONFIG : 'N U T, 0, 0, 0',
    X =  451.279  mm,    Y =   18.682  mm,    Z =   -319.944  mm,
    W =  -188.998 deg,    P =   0.156 deg,    R =   -0.986 deg
};
P[78]{
   GP1:
    UF : 0, UT : 6,      CONFIG : 'N U T, 0, 0, 0',
    X =  454.203  mm,    Y =   17.068  mm,    Z =   -317.405  mm,
    W =  -188.912 deg,    P =   0.155 deg,    R =   -0.986 deg
};
P[79]{
   GP1:
    UF : 0, UT : 6,      CONFIG : 'N U T, 0, 0, 0',
    X =  451.974  mm,    Y =   13.360  mm,    Z =   -314.280  mm,
    W =  -188.962 deg,    P =   0.156 deg,    R =   -0.986 deg
};
P[80]{
   GP1:
    UF : 0, UT : 6,      CONFIG : 'N U T, 0, 0, 0',
    X =  451.186  mm,    Y =   4.148  mm,    Z =   -305.021  mm,
    W =  -188.772 deg,    P =   0.152 deg,    R =   -0.987 deg
};
P[81]{
   GP1:
    UF : 0, UT : 6,      CONFIG : 'N U T, 0, 0, 0',
    X =  451.854  mm,    Y =   -1.076  mm,    Z =   -299.304  mm,
    W =  -188.639 deg,    P =   0.150 deg,    R =   -0.988 deg
};
P[82]{
   GP1:
    UF : 0, UT : 6,      CONFIG : 'N U T, 0, 0, 0',
    X =  451.123  mm,    Y =   -5.563  mm,    Z =   -294.706  mm,
    W =  -188.579 deg,    P =   0.149 deg,    R =   -0.988 deg
};
P[83]{
   GP1:
    UF : 0, UT : 6,      CONFIG : 'N U T, 0, 0, 0',
    X =  454.573  mm,    Y =   -6.529  mm,    Z =   -293.143  mm,
    W =  -188.646 deg,    P =   0.150 deg,    R =   -0.987 deg
};
P[84]{
   GP1:
    UF : 0, UT : 6,      CONFIG : 'N U T, 0, 0, 0',
    X =  451.093  mm,    Y =   -10.889  mm,    Z =   -289.987  mm,
    W =  -188.511 deg,    P =   0.148 deg,    R =   -0.988 deg
};
P[85]{
   GP1:
    UF : 0, UT : 6,      CONFIG : 'N U T, 0, 0, 0',
    X =  451.219  mm,    Y =   -16.052  mm,    Z =   -290.165  mm,
    W =  -188.450 deg,    P =   0.147 deg,    R =   -0.988 deg
};
P[86]{
   GP1:
    UF : 0, UT : 6,      CONFIG : 'N U T, 0, 0, 0',
    X =  451.073  mm,    Y =   -21.515  mm,    Z =   -290.824  mm,
    W =  -188.344 deg,    P =   0.145 deg,    R =   -0.988 deg
};
P[87]{
   GP1:
    UF : 0, UT : 6,      CONFIG : 'N U T, 0, 0, 0',
    X =  453.779  mm,    Y =   -25.228  mm,    Z =   -291.194  mm,
    W =  -188.373 deg,    P =   0.145 deg,    R =   -0.988 deg
};
P[88]{
   GP1:
    UF : 0, UT : 6,      CONFIG : 'N U T, 0, 0, 0',
    X =  451.290  mm,    Y =   -26.832  mm,    Z =   -291.575  mm,
    W =  -188.337 deg,    P =   0.145 deg,    R =   -0.988 deg
};
P[89]{
   GP1:
    UF : 0, UT : 6,      CONFIG : 'N U T, 0, 0, 0',
    X =  451.254  mm,    Y =   -33.249  mm,    Z =   -294.009  mm,
    W =  -188.199 deg,    P =   0.142 deg,    R =   -0.988 deg
};
P[90]{
   GP1:
    UF : 0, UT : 6,      CONFIG : 'N U T, 0, 0, 0',
    X =  450.801  mm,    Y =   -37.492  mm,    Z =   -308.406  mm,
    W =  -188.263 deg,    P =   0.144 deg,    R =   -0.988 deg
};
P[91]{
   GP1:
    UF : 0, UT : 6,      CONFIG : 'N U T, 0, 0, 0',
    X =  451.209  mm,    Y =   -41.802  mm,    Z =   -308.406  mm,
    W =  -188.309 deg,    P =   0.144 deg,    R =   -0.988 deg
};
P[92]{
   GP1:
    UF : 0, UT : 6,      CONFIG : 'N U T, 0, 0, 0',
    X =  452.568  mm,    Y =   -45.042  mm,    Z =   -308.406  mm,
    W =  -188.205 deg,    P =   0.142 deg,    R =   -0.988 deg
};
P[93]{
   GP1:
    UF : 0, UT : 6,      CONFIG : 'N U T, 0, 0, 0',
    X =  451.143  mm,    Y =   -45.969  mm,    Z =   -308.406  mm,
    W =  -188.083 deg,    P =   0.140 deg,    R =   -0.988 deg
};
P[94]{
   GP1:
    UF : 0, UT : 6,      CONFIG : 'N U T, 0, 0, 0',
    X =  451.122  mm,    Y =   -46.680  mm,    Z =   -308.406  mm,
    W =  -188.130 deg,    P =   0.141 deg,    R =   -0.988 deg
};
P[95]{
   GP1:
    UF : 0, UT : 6,      CONFIG : 'N U T, 0, 0, 0',
    X =  450.939  mm,    Y =   -46.713  mm,    Z =   -308.406  mm,
    W =  -188.215 deg,    P =   0.143 deg,    R =   -0.988 deg
};
P[96]{
   GP1:
    UF : 0, UT : 6,      CONFIG : 'N U T, 0, 0, 0',
    X =  452.878  mm,    Y =   -95.475  mm,    Z =   -325.827  mm,
    W =  -180.000 deg,    P =   0.000 deg,    R =   0.000 deg
};
P[97]{
   GP1:
    UF : 0, UT : 6,      CONFIG : 'N U T, 0, 0, 0',
    X =  426.439  mm,    Y =   -95.475  mm,    Z =   -325.827  mm,
    W =  -180.000 deg,    P =   0.000 deg,    R =   0.000 deg
};
P[98]{
   GP1:
    UF : 0, UT : 6,      CONFIG : 'N U T, 0, 0, 0',
    X =  426.504  mm,    Y =   -41.584  mm,    Z =   -324.704  mm,
    W =  -186.470 deg,    P =   0.113 deg,    R =   -0.993 deg
};
P[99]{
   GP1:
    UF : 0, UT : 6,      CONFIG : 'N U T, 0, 0, 0',
    X =  425.902  mm,    Y =   -39.793  mm,    Z =   -324.704  mm,
    W =  -186.558 deg,    P =   0.114 deg,    R =   -0.993 deg
};
P[100]{
   GP1:
    UF : 0, UT : 6,      CONFIG : 'N U T, 0, 0, 0',
    X =  426.059  mm,    Y =   -37.192  mm,    Z =   -324.704  mm,
    W =  -186.639 deg,    P =   0.116 deg,    R =   -0.993 deg
};
P[101]{
   GP1:
    UF : 0, UT : 6,      CONFIG : 'N U T, 0, 0, 0',
    X =  426.850  mm,    Y =   -34.445  mm,    Z =   -324.704  mm,
    W =  -186.739 deg,    P =   0.117 deg,    R =   -0.993 deg
};
P[102]{
   GP1:
    UF : 0, UT : 6,      CONFIG : 'N U T, 0, 0, 0',
    X =  426.148  mm,    Y =   -31.859  mm,    Z =   -302.734  mm,
    W =  -186.837 deg,    P =   0.119 deg,    R =   -0.993 deg
};
P[103]{
   GP1:
    UF : 0, UT : 6,      CONFIG : 'N U T, 0, 0, 0',
    X =  425.989  mm,    Y =   -27.561  mm,    Z =   -299.877  mm,
    W =  -186.967 deg,    P =   0.121 deg,    R =   -0.992 deg
};
P[104]{
   GP1:
    UF : 0, UT : 6,      CONFIG : 'N U T, 0, 0, 0',
    X =  426.968  mm,    Y =   -23.153  mm,    Z =   -300.283  mm,
    W =  -187.047 deg,    P =   0.123 deg,    R =   -0.992 deg
};
P[105]{
   GP1:
    UF : 0, UT : 6,      CONFIG : 'N U T, 0, 0, 0',
    X =  425.990  mm,    Y =   -20.515  mm,    Z =   -301.308  mm,
    W =  -187.103 deg,    P =   0.124 deg,    R =   -0.992 deg
};
P[106]{
   GP1:
    UF : 0, UT : 6,      CONFIG : 'N U T, 0, 0, 0',
    X =  425.920  mm,    Y =   -14.693  mm,    Z =   -302.160  mm,
    W =  -187.196 deg,    P =   0.125 deg,    R =   -0.992 deg
};
P[107]{
   GP1:
    UF : 0, UT : 6,      CONFIG : 'N U T, 0, 0, 0',
    X =  425.963  mm,    Y =   -9.572  mm,    Z =   -301.494  mm,
    W =  -187.301 deg,    P =   0.127 deg,    R =   -0.992 deg
};
P[108]{
   GP1:
    UF : 0, UT : 6,      CONFIG : 'N U T, 0, 0, 0',
    X =  426.559  mm,    Y =   -3.508  mm,    Z =   -305.015  mm,
    W =  -187.520 deg,    P =   0.131 deg,    R =   -0.991 deg
};
P[109]{
   GP1:
    UF : 0, UT : 6,      CONFIG : 'N U T, 0, 0, 0',
    X =  427.257  mm,    Y =   1.808  mm,    Z =   -308.672  mm,
    W =  -187.710 deg,    P =   0.134 deg,    R =   -0.991 deg
};
P[110]{
   GP1:
    UF : 0, UT : 6,      CONFIG : 'N U T, 0, 0, 0',
    X =  424.606  mm,    Y =   3.260  mm,    Z =   -311.722  mm,
    W =  -187.552 deg,    P =   0.131 deg,    R =   -0.991 deg
};
P[111]{
   GP1:
    UF : 0, UT : 6,      CONFIG : 'N U T, 0, 0, 0',
    X =  426.816  mm,    Y =   7.202  mm,    Z =   -313.307  mm,
    W =  -187.865 deg,    P =   0.137 deg,    R =   -0.990 deg
};
P[112]{
   GP1:
    UF : 0, UT : 6,      CONFIG : 'N U T, 0, 0, 0',
    X =  426.388  mm,    Y =   12.117  mm,    Z =   -317.772  mm,
    W =  -188.097 deg,    P =   0.141 deg,    R =   -0.989 deg
};
P[113]{
   GP1:
    UF : 0, UT : 6,      CONFIG : 'N U T, 0, 0, 0',
    X =  427.777  mm,    Y =   14.475  mm,    Z =   -318.783  mm,
    W =  -188.177 deg,    P =   0.142 deg,    R =   -0.989 deg
};
P[114]{
   GP1:
    UF : 0, UT : 6,      CONFIG : 'N U T, 0, 0, 0',
    X =  425.572  mm,    Y =   16.123  mm,    Z =   -321.399  mm,
    W =  -188.164 deg,    P =   0.142 deg,    R =   -0.989 deg
};
P[115]{
   GP1:
    UF : 0, UT : 6,      CONFIG : 'N U T, 0, 0, 0',
    X =  426.030  mm,    Y =   20.610  mm,    Z =   -302.922  mm,
    W =  -187.914 deg,    P =   0.138 deg,    R =   -0.990 deg
};
P[116]{
   GP1:
    UF : 0, UT : 6,      CONFIG : 'N U T, 0, 0, 0',
    X =  426.319  mm,    Y =   20.921  mm,    Z =   -308.183  mm,
    W =  -188.008 deg,    P =   0.139 deg,    R =   -0.989 deg
};
P[117]{
   GP1:
    UF : 0, UT : 6,      CONFIG : 'N U T, 0, 0, 0',
    X =  425.862  mm,    Y =   21.461  mm,    Z =   -319.373  mm,
    W =  -188.194 deg,    P =   0.142 deg,    R =   -0.989 deg
};
P[118]{
   GP1:
    UF : 0, UT : 6,      CONFIG : 'N U T, 0, 0, 0',
    X =  424.513  mm,    Y =   21.566  mm,    Z =   -323.791  mm,
    W =  -188.210 deg,    P =   0.143 deg,    R =   -0.989 deg
};
P[119]{
   GP1:
    UF : 0, UT : 6,      CONFIG : 'N U T, 0, 0, 0',
    X =  425.886  mm,    Y =   21.598  mm,    Z =   -313.203  mm,
    W =  -188.110 deg,    P =   0.141 deg,    R =   -0.989 deg
};
P[120]{
   GP1:
    UF : 0, UT : 6,      CONFIG : 'N U T, 0, 0, 0',
    X =  426.108  mm,    Y =   22.735  mm,    Z =   -299.668  mm,
    W =  -187.993 deg,    P =   0.139 deg,    R =   -0.989 deg
};
P[121]{
   GP1:
    UF : 0, UT : 6,      CONFIG : 'N U T, 0, 0, 0',
    X =  426.041  mm,    Y =   28.094  mm,    Z =   -298.659  mm,
    W =  -187.966 deg,    P =   0.138 deg,    R =   -0.989 deg
};
P[122]{
   GP1:
    UF : 0, UT : 6,      CONFIG : 'N U T, 0, 0, 0',
    X =  425.944  mm,    Y =   32.633  mm,    Z =   -298.935  mm,
    W =  -188.123 deg,    P =   0.141 deg,    R =   -0.989 deg
};
P[123]{
   GP1:
    UF : 0, UT : 6,      CONFIG : 'N U T, 0, 0, 0',
    X =  425.893  mm,    Y =   35.270  mm,    Z =   -298.949  mm,
    W =  -188.037 deg,    P =   0.140 deg,    R =   -0.989 deg
};
P[124]{
   GP1:
    UF : 0, UT : 6,      CONFIG : 'N U T, 0, 0, 0',
    X =  426.537  mm,    Y =   39.619  mm,    Z =   -298.871  mm,
    W =  -187.811 deg,    P =   0.136 deg,    R =   -0.989 deg
};
P[125]{
   GP1:
    UF : 0, UT : 6,      CONFIG : 'N U T, 0, 0, 0',
    X =  426.124  mm,    Y =   46.679  mm,    Z =   -303.015  mm,
    W =  -186.860 deg,    P =   0.119 deg,    R =   -0.991 deg
};
P[126]{
   GP1:
    UF : 0, UT : 6,      CONFIG : 'N U T, 0, 0, 0',
    X =  426.135  mm,    Y =   53.362  mm,    Z =   -303.015  mm,
    W =  -185.679 deg,    P =   0.099 deg,    R =   -0.993 deg
};
P[127]{
   GP1:
    UF : 0, UT : 6,      CONFIG : 'N U T, 0, 0, 0',
    X =  426.439  mm,    Y =   95.475  mm,    Z =   -325.827  mm,
    W =  -180.000 deg,    P =   0.000 deg,    R =   0.000 deg
};
P[128]{
   GP1:
    UF : 0, UT : 6,      CONFIG : 'N U T, 0, 0, 0',
    X =  400.000  mm,    Y =   95.475  mm,    Z =   -325.827  mm,
    W =  -180.000 deg,    P =   0.000 deg,    R =   0.000 deg
};
P[129]{
   GP1:
    UF : 0, UT : 6,      CONFIG : 'N U T, 0, 0, 0',
    X =  401.353  mm,    Y =   52.067  mm,    Z =   -298.795  mm,
    W =  -186.919 deg,    P =   0.120 deg,    R =   -0.993 deg
};
P[130]{
   GP1:
    UF : 0, UT : 6,      CONFIG : 'N U T, 0, 0, 0',
    X =  400.579  mm,    Y =   45.987  mm,    Z =   -298.795  mm,
    W =  -186.490 deg,    P =   0.113 deg,    R =   -0.994 deg
};
P[131]{
   GP1:
    UF : 0, UT : 6,      CONFIG : 'N U T, 0, 0, 0',
    X =  401.361  mm,    Y =   41.768  mm,    Z =   -291.814  mm,
    W =  -186.622 deg,    P =   0.115 deg,    R =   -0.993 deg
};
P[132]{
   GP1:
    UF : 0, UT : 6,      CONFIG : 'N U T, 0, 0, 0',
    X =  401.045  mm,    Y =   36.105  mm,    Z =   -292.087  mm,
    W =  -186.389 deg,    P =   0.111 deg,    R =   -0.994 deg
};
P[133]{
   GP1:
    UF : 0, UT : 6,      CONFIG : 'N U T, 0, 0, 0',
    X =  401.110  mm,    Y =   31.559  mm,    Z =   -293.655  mm,
    W =  -186.420 deg,    P =   0.112 deg,    R =   -0.994 deg
};
P[134]{
   GP1:
    UF : 0, UT : 6,      CONFIG : 'N U T, 0, 0, 0',
    X =  401.182  mm,    Y =   26.660  mm,    Z =   -295.316  mm,
    W =  -186.411 deg,    P =   0.112 deg,    R =   -0.994 deg
};
P[135]{
   GP1:
    UF : 0, UT : 6,      CONFIG : 'N U T, 0, 0, 0',
    X =  401.182  mm,    Y =   22.244  mm,    Z =   -297.664  mm,
    W =  -186.371 deg,    P =   0.111 deg,    R =   -0.994 deg
};
P[136]{
   GP1:
    UF : 0, UT : 6,      CONFIG : 'N U T, 0, 0, 0',
    X =  401.318  mm,    Y =   18.262  mm,    Z =   -300.348  mm,
    W =  -186.342 deg,    P =   0.110 deg,    R =   -0.994 deg
};
P[137]{
   GP1:
    UF : 0, UT : 6,      CONFIG : 'N U T, 0, 0, 0',
    X =  400.548  mm,    Y =   16.657  mm,    Z =   -304.245  mm,
    W =  -186.526 deg,    P =   0.114 deg,    R =   -0.994 deg
};
P[138]{
   GP1:
    UF : 0, UT : 6,      CONFIG : 'N U T, 0, 0, 0',
    X =  400.726  mm,    Y =   16.442  mm,    Z =   -310.489  mm,
    W =  -186.540 deg,    P =   0.114 deg,    R =   -0.993 deg
};
P[139]{
   GP1:
    UF : 0, UT : 6,      CONFIG : 'N U T, 0, 0, 0',
    X =  401.625  mm,    Y =   13.094  mm,    Z =   -312.810  mm,
    W =  -186.625 deg,    P =   0.115 deg,    R =   -0.993 deg
};
P[140]{
   GP1:
    UF : 0, UT : 6,      CONFIG : 'N U T, 0, 0, 0',
    X =  401.290  mm,    Y =   6.666  mm,    Z =   -310.855  mm,
    W =  -186.521 deg,    P =   0.114 deg,    R =   -0.994 deg
};
P[141]{
   GP1:
    UF : 0, UT : 6,      CONFIG : 'N U T, 0, 0, 0',
    X =  401.282  mm,    Y =   1.445  mm,    Z =   -307.402  mm,
    W =  -186.556 deg,    P =   0.114 deg,    R =   -0.993 deg
};
P[142]{
   GP1:
    UF : 0, UT : 6,      CONFIG : 'N U T, 0, 0, 0',
    X =  400.467  mm,    Y =   -4.013  mm,    Z =   -302.564  mm,
    W =  -186.575 deg,    P =   0.115 deg,    R =   -0.993 deg
};
P[143]{
   GP1:
    UF : 0, UT : 6,      CONFIG : 'N U T, 0, 0, 0',
    X =  401.488  mm,    Y =   -7.685  mm,    Z =   -301.726  mm,
    W =  -186.610 deg,    P =   0.115 deg,    R =   -0.993 deg
};
P[144]{
   GP1:
    UF : 0, UT : 6,      CONFIG : 'N U T, 0, 0, 0',
    X =  401.392  mm,    Y =   -14.205  mm,    Z =   -303.858  mm,
    W =  -186.611 deg,    P =   0.115 deg,    R =   -0.993 deg
};
P[145]{
   GP1:
    UF : 0, UT : 6,      CONFIG : 'N U T, 0, 0, 0',
    X =  401.836  mm,    Y =   -18.733  mm,    Z =   -303.798  mm,
    W =  -186.589 deg,    P =   0.115 deg,    R =   -0.993 deg
};
P[146]{
   GP1:
    UF : 0, UT : 6,      CONFIG : 'N U T, 0, 0, 0',
    X =  400.869  mm,    Y =   -24.118  mm,    Z =   -302.307  mm,
    W =  -186.596 deg,    P =   0.115 deg,    R =   -0.993 deg
};
P[147]{
   GP1:
    UF : 0, UT : 6,      CONFIG : 'N U T, 0, 0, 0',
    X =  399.952  mm,    Y =   -28.147  mm,    Z =   -302.498  mm,
    W =  -186.585 deg,    P =   0.115 deg,    R =   -0.993 deg
};
P[148]{
   GP1:
    UF : 0, UT : 6,      CONFIG : 'N U T, 0, 0, 0',
    X =  401.173  mm,    Y =   -29.947  mm,    Z =   -307.407  mm,
    W =  -186.545 deg,    P =   0.114 deg,    R =   -0.993 deg
};
P[149]{
   GP1:
    UF : 0, UT : 6,      CONFIG : 'N U T, 0, 0, 0',
    X =  401.309  mm,    Y =   -32.001  mm,    Z =   -313.225  mm,
    W =  -186.448 deg,    P =   0.112 deg,    R =   -0.994 deg
};
P[150]{
   GP1:
    UF : 0, UT : 6,      CONFIG : 'N U T, 0, 0, 0',
    X =  401.098  mm,    Y =   -34.386  mm,    Z =   -322.998  mm,
    W =  -186.423 deg,    P =   0.112 deg,    R =   -0.994 deg
};
P[151]{
   GP1:
    UF : 0, UT : 6,      CONFIG : 'N U T, 0, 0, 0',
    X =  402.041  mm,    Y =   -38.612  mm,    Z =   -322.998  mm,
    W =  -186.293 deg,    P =   0.110 deg,    R =   -0.994 deg
};
P[152]{
   GP1:
    UF : 0, UT : 6,      CONFIG : 'N U T, 0, 0, 0',
    X =  399.502  mm,    Y =   -39.593  mm,    Z =   -322.998  mm,
    W =  -186.235 deg,    P =   0.109 deg,    R =   -0.994 deg
};
P[153]{
   GP1:
    UF : 0, UT : 6,      CONFIG : 'N U T, 0, 0, 0',
    X =  401.212  mm,    Y =   -43.375  mm,    Z =   -322.998  mm,
    W =  -186.143 deg,    P =   0.107 deg,    R =   -0.994 deg
};
P[154]{
   GP1:
    UF : 0, UT : 6,      CONFIG : 'N U T, 0, 0, 0',
    X =  400.000  mm,    Y =   -95.475  mm,    Z =   -325.827  mm,
    W =  -180.000 deg,    P =   0.000 deg,    R =   0.000 deg
};
P[155]{
   GP1:
    UF : 0, UT : 6,      CONFIG : 'N U T, 0, 0, 0',
    X =  373.561  mm,    Y =   -95.475  mm,    Z =   -325.827  mm,
    W =  -180.000 deg,    P =   0.000 deg,    R =   0.000 deg
};
P[156]{
   GP1:
    UF : 0, UT : 6,      CONFIG : 'N U T, 0, 0, 0',
    X =  371.600  mm,    Y =   -38.825  mm,    Z =   -321.075  mm,
    W =  -187.535 deg,    P =   0.131 deg,    R =   -0.991 deg
};
P[157]{
   GP1:
    UF : 0, UT : 6,      CONFIG : 'N U T, 0, 0, 0',
    X =  371.546  mm,    Y =   -30.350  mm,    Z =   -321.075  mm,
    W =  -186.852 deg,    P =   0.119 deg,    R =   -0.993 deg
};
P[158]{
   GP1:
    UF : 0, UT : 6,      CONFIG : 'N U T, 0, 0, 0',
    X =  371.726  mm,    Y =   -24.167  mm,    Z =   -302.408  mm,
    W =  -186.822 deg,    P =   0.119 deg,    R =   -0.993 deg
};
P[159]{
   GP1:
    UF : 0, UT : 6,      CONFIG : 'N U T, 0, 0, 0',
    X =  375.001  mm,    Y =   -23.849  mm,    Z =   -305.121  mm,
    W =  -186.789 deg,    P =   0.118 deg,    R =   -0.993 deg
};
P[160]{
   GP1:
    UF : 0, UT : 6,      CONFIG : 'N U T, 0, 0, 0',
    X =  371.403  mm,    Y =   -7.657  mm,    Z =   -306.059  mm,
    W =  -186.577 deg,    P =   0.115 deg,    R =   -0.993 deg
};
P[161]{
   GP1:
    UF : 0, UT : 6,      CONFIG : 'N U T, 0, 0, 0',
    X =  371.713  mm,    Y =   2.306  mm,    Z =   -305.228  mm,
    W =  -186.257 deg,    P =   0.109 deg,    R =   -0.994 deg
};
P[162]{
   GP1:
    UF : 0, UT : 6,      CONFIG : 'N U T, 0, 0, 0',
    X =  371.585  mm,    Y =   11.006  mm,    Z =   -306.093  mm,
    W =  -185.752 deg,    P =   0.100 deg,    R =   -0.995 deg
};
P[163]{
   GP1:
    UF : 0, UT : 6,      CONFIG : 'N U T, 0, 0, 0',
    X =  371.387  mm,    Y =   14.734  mm,    Z =   -305.715  mm,
    W =  -185.590 deg,    P =   0.097 deg,    R =   -0.995 deg
};
P[164]{
   GP1:
    UF : 0, UT : 6,      CONFIG : 'N U T, 0, 0, 0',
    X =  375.413  mm,    Y =   30.564  mm,    Z =   -301.310  mm,
    W =  -185.287 deg,    P =   0.092 deg,    R =   -0.996 deg
};
P[165]{
   GP1:
    UF : 0, UT : 6,      CONFIG : 'N U T, 0, 0, 0',
    X =  375.748  mm,    Y =   41.563  mm,    Z =   -297.255  mm,
    W =  -185.012 deg,    P =   0.087 deg,    R =   -0.996 deg
};
P[166]{
   GP1:
    UF : 0, UT : 6,      CONFIG : 'N U T, 0, 0, 0',
    X =  373.561  mm,    Y =   95.475  mm,    Z =   -325.827  mm,
    W =  -180.000 deg,    P =   0.000 deg,    R =   0.000 deg
};
P[167]{
   GP1:
    UF : 0, UT : 6,      CONFIG : 'N U T, 0, 0, 0',
    X =  347.122  mm,    Y =   95.475  mm,    Z =   -325.827  mm,
    W =  -180.000 deg,    P =   0.000 deg,    R =   0.000 deg
};
P[168]{
   GP1:
    UF : 0, UT : 6,      CONFIG : 'N U T, 0, 0, 0',
    X =  346.516  mm,    Y =   31.645  mm,    Z =   -294.025  mm,
    W =  -182.787 deg,    P =   0.049 deg,    R =   -0.999 deg
};
P[169]{
   GP1:
    UF : 0, UT : 6,      CONFIG : 'N U T, 0, 0, 0',
    X =  346.354  mm,    Y =   26.090  mm,    Z =   -294.025  mm,
    W =  -183.177 deg,    P =   0.055 deg,    R =   -0.998 deg
};
P[170]{
   GP1:
    UF : 0, UT : 6,      CONFIG : 'N U T, 0, 0, 0',
    X =  346.553  mm,    Y =   21.085  mm,    Z =   -295.945  mm,
    W =  -183.328 deg,    P =   0.058 deg,    R =   -0.998 deg
};
P[171]{
   GP1:
    UF : 0, UT : 6,      CONFIG : 'N U T, 0, 0, 0',
    X =  346.495  mm,    Y =   16.857  mm,    Z =   -298.546  mm,
    W =  -183.574 deg,    P =   0.062 deg,    R =   -0.998 deg
};
P[172]{
   GP1:
    UF : 0, UT : 6,      CONFIG : 'N U T, 0, 0, 0',
    X =  345.951  mm,    Y =   11.119  mm,    Z =   -300.229  mm,
    W =  -183.774 deg,    P =   0.066 deg,    R =   -0.997 deg
};
P[173]{
   GP1:
    UF : 0, UT : 6,      CONFIG : 'N U T, 0, 0, 0',
    X =  346.050  mm,    Y =   5.703  mm,    Z =   -299.767  mm,
    W =  -183.952 deg,    P =   0.069 deg,    R =   -0.997 deg
};
P[174]{
   GP1:
    UF : 0, UT : 6,      CONFIG : 'N U T, 0, 0, 0',
    X =  346.147  mm,    Y =   0.857  mm,    Z =   -299.353  mm,
    W =  -184.089 deg,    P =   0.071 deg,    R =   -0.997 deg
};
P[175]{
   GP1:
    UF : 0, UT : 6,      CONFIG : 'N U T, 0, 0, 0',
    X =  346.113  mm,    Y =   -5.664  mm,    Z =   -298.825  mm,
    W =  -184.337 deg,    P =   0.076 deg,    R =   -0.997 deg
};
P[176]{
   GP1:
    UF : 0, UT : 6,      CONFIG : 'N U T, 0, 0, 0',
    X =  346.092  mm,    Y =   -13.425  mm,    Z =   -297.633  mm,
    W =  -185.406 deg,    P =   0.094 deg,    R =   -0.995 deg
};
P[177]{
   GP1:
    UF : 0, UT : 6,      CONFIG : 'N U T, 0, 0, 0',
    X =  346.016  mm,    Y =   -19.033  mm,    Z =   -296.651  mm,
    W =  -186.083 deg,    P =   0.106 deg,    R =   -0.994 deg
};
P[178]{
   GP1:
    UF : 0, UT : 6,      CONFIG : 'N U T, 0, 0, 0',
    X =  346.555  mm,    Y =   -24.417  mm,    Z =   -295.632  mm,
    W =  -186.737 deg,    P =   0.117 deg,    R =   -0.993 deg
};
P[179]{
   GP1:
    UF : 0, UT : 6,      CONFIG : 'N U T, 0, 0, 0',
    X =  345.946  mm,    Y =   -29.979  mm,    Z =   -295.580  mm,
    W =  -187.144 deg,    P =   0.124 deg,    R =   -0.992 deg
};
P[180]{
   GP1:
    UF : 0, UT : 6,      CONFIG : 'N U T, 0, 0, 0',
    X =  346.628  mm,    Y =   -34.224  mm,    Z =   -296.139  mm,
    W =  -187.475 deg,    P =   0.130 deg,    R =   -0.991 deg
};
P[181]{
   GP1:
    UF : 0, UT : 6,      CONFIG : 'N U T, 0, 0, 0',
    X =  346.050  mm,    Y =   -38.739  mm,    Z =   -296.458  mm,
    W =  -187.948 deg,    P =   0.138 deg,    R =   -0.990 deg
};
P[182]{
   GP1:
    UF : 0, UT : 6,      CONFIG : 'N U T, 0, 0, 0',
    X =  346.529  mm,    Y =   -45.280  mm,    Z =   -297.929  mm,
    W =  -188.242 deg,    P =   0.143 deg,    R =   -0.990 deg
};
P[183]{
   GP1:
    UF : 0, UT : 6,      CONFIG : 'N U T, 0, 0, 0',
    X =  346.228  mm,    Y =   -50.704  mm,    Z =   -312.069  mm,
    W =  -188.458 deg,    P =   0.147 deg,    R =   -0.989 deg
};
P[184]{
   GP1:
    UF : 0, UT : 6,      CONFIG : 'N U T, 0, 0, 0',
    X =  346.206  mm,    Y =   -54.809  mm,    Z =   -312.069  mm,
    W =  -188.704 deg,    P =   0.151 deg,    R =   -0.988 deg
};
P[185]{
   GP1:
    UF : 0, UT : 6,      CONFIG : 'N U T, 0, 0, 0',
    X =  346.213  mm,    Y =   -56.991  mm,    Z =   -312.069  mm,
    W =  -188.797 deg,    P =   0.153 deg,    R =   -0.988 deg
};
P[186]{
   GP1:
    UF : 0, UT : 6,      CONFIG : 'N U T, 0, 0, 0',
    X =  346.193  mm,    Y =   -57.982  mm,    Z =   -312.069  mm,
    W =  -188.932 deg,    P =   0.155 deg,    R =   -0.988 deg
};
P[187]{
   GP1:
    UF : 0, UT : 6,      CONFIG : 'N U T, 0, 0, 0',
    X =  346.156  mm,    Y =   -57.989  mm,    Z =   -312.069  mm,
    W =  -188.826 deg,    P =   0.153 deg,    R =   -0.988 deg
};
P[188]{
   GP1:
    UF : 0, UT : 6,      CONFIG : 'N U T, 0, 0, 0',
    X =  346.264  mm,    Y =   -58.816  mm,    Z =   -312.069  mm,
    W =  -188.993 deg,    P =   0.156 deg,    R =   -0.988 deg
};
P[189]{
   GP1:
    UF : 0, UT : 6,      CONFIG : 'N U T, 0, 0, 0',
    X =  345.824  mm,    Y =   -59.164  mm,    Z =   -312.069  mm,
    W =  -189.023 deg,    P =   0.157 deg,    R =   -0.988 deg
};
P[190]{
   GP1:
    UF : 0, UT : 6,      CONFIG : 'N U T, 0, 0, 0',
    X =  347.122  mm,    Y =   -95.475  mm,    Z =   -325.827  mm,
    W =  -180.000 deg,    P =   0.000 deg,    R =   0.000 deg
};
P[191]{
   GP1:
    UF : 0, UT : 6,      CONFIG : 'N U T, 0, 0, 0',
    X =  320.683  mm,    Y =   -95.475  mm,    Z =   -325.827  mm,
    W =  -180.000 deg,    P =   0.000 deg,    R =   0.000 deg
};
P[192]{
   GP1:
    UF : 0, UT : 6,      CONFIG : 'N U T, 0, 0, 0',
    X =  321.273  mm,    Y =   -63.653  mm,    Z =   -319.364  mm,
    W =  -189.449 deg,    P =   0.164 deg,    R =   -0.986 deg
};
P[193]{
   GP1:
    UF : 0, UT : 6,      CONFIG : 'N U T, 0, 0, 0',
    X =  321.334  mm,    Y =   -63.456  mm,    Z =   -319.364  mm,
    W =  -189.401 deg,    P =   0.163 deg,    R =   -0.986 deg
};
P[194]{
   GP1:
    UF : 0, UT : 6,      CONFIG : 'N U T, 0, 0, 0',
    X =  322.582  mm,    Y =   -62.926  mm,    Z =   -319.364  mm,
    W =  -189.432 deg,    P =   0.164 deg,    R =   -0.986 deg
};
P[195]{
   GP1:
    UF : 0, UT : 6,      CONFIG : 'N U T, 0, 0, 0',
    X =  320.688  mm,    Y =   -61.711  mm,    Z =   -319.364  mm,
    W =  -189.180 deg,    P =   0.159 deg,    R =   -0.986 deg
};
P[196]{
   GP1:
    UF : 0, UT : 6,      CONFIG : 'N U T, 0, 0, 0',
    X =  321.911  mm,    Y =   -58.656  mm,    Z =   -319.364  mm,
    W =  -188.856 deg,    P =   0.154 deg,    R =   -0.987 deg
};
P[197]{
   GP1:
    UF : 0, UT : 6,      CONFIG : 'N U T, 0, 0, 0',
    X =  321.062  mm,    Y =   -54.532  mm,    Z =   -319.364  mm,
    W =  -188.306 deg,    P =   0.144 deg,    R =   -0.989 deg
};
P[198]{
   GP1:
    UF : 0, UT : 6,      CONFIG : 'N U T, 0, 0, 0',
    X =  320.969  mm,    Y =   -49.972  mm,    Z =   -300.882  mm,
    W =  -187.474 deg,    P =   0.130 deg,    R =   -0.990 deg
};
P[199]{
   GP1:
    UF : 0, UT : 6,      CONFIG : 'N U T, 0, 0, 0',
    X =  320.866  mm,    Y =   -43.532  mm,    Z =   -299.793  mm,
    W =  -186.521 deg,    P =   0.113 deg,    R =   -0.992 deg
};
P[200]{
   GP1:
    UF : 0, UT : 6,      CONFIG : 'N U T, 0, 0, 0',
    X =  321.050  mm,    Y =   -38.839  mm,    Z =   -299.975  mm,
    W =  -185.952 deg,    P =   0.104 deg,    R =   -0.993 deg
};
P[201]{
   GP1:
    UF : 0, UT : 6,      CONFIG : 'N U T, 0, 0, 0',
    X =  321.852  mm,    Y =   -34.723  mm,    Z =   -300.206  mm,
    W =  -185.571 deg,    P =   0.097 deg,    R =   -0.994 deg
};
P[202]{
   GP1:
    UF : 0, UT : 6,      CONFIG : 'N U T, 0, 0, 0',
    X =  320.413  mm,    Y =   -31.666  mm,    Z =   -301.035  mm,
    W =  -184.971 deg,    P =   0.087 deg,    R =   -0.995 deg
};
P[203]{
   GP1:
    UF : 0, UT : 6,      CONFIG : 'N U T, 0, 0, 0',
    X =  320.938  mm,    Y =   -27.005  mm,    Z =   -300.066  mm,
    W =  -184.640 deg,    P =   0.081 deg,    R =   -0.995 deg
};
P[204]{
   GP1:
    UF : 0, UT : 6,      CONFIG : 'N U T, 0, 0, 0',
    X =  321.877  mm,    Y =   -22.780  mm,    Z =   -298.952  mm,
    W =  -184.336 deg,    P =   0.075 deg,    R =   -0.995 deg
};
P[205]{
   GP1:
    UF : 0, UT : 6,      CONFIG : 'N U T, 0, 0, 0',
    X =  320.812  mm,    Y =   -18.094  mm,    Z =   -299.859  mm,
    W =  -184.282 deg,    P =   0.075 deg,    R =   -0.995 deg
};
P[206]{
   GP1:
    UF : 0, UT : 6,      CONFIG : 'N U T, 0, 0, 0',
    X =  322.326  mm,    Y =   -12.063  mm,    Z =   -300.049  mm,
    W =  -184.315 deg,    P =   0.075 deg,    R =   -0.995 deg
};
P[207]{
   GP1:
    UF : 0, UT : 6,      CONFIG : 'N U T, 0, 0, 0',
    X =  321.090  mm,    Y =   -9.745  mm,    Z =   -300.435  mm,
    W =  -184.250 deg,    P =   0.074 deg,    R =   -0.995 deg
};
P[208]{
   GP1:
    UF : 0, UT : 6,      CONFIG : 'N U T, 0, 0, 0',
    X =  320.896  mm,    Y =   -4.915  mm,    Z =   -299.741  mm,
    W =  -184.118 deg,    P =   0.072 deg,    R =   -0.996 deg
};
P[209]{
   GP1:
    UF : 0, UT : 6,      CONFIG : 'N U T, 0, 0, 0',
    X =  321.201  mm,    Y =   0.590  mm,    Z =   -299.721  mm,
    W =  -184.035 deg,    P =   0.070 deg,    R =   -0.996 deg
};
P[210]{
   GP1:
    UF : 0, UT : 6,      CONFIG : 'N U T, 0, 0, 0',
    X =  321.088  mm,    Y =   5.888  mm,    Z =   -299.817  mm,
    W =  -183.914 deg,    P =   0.068 deg,    R =   -0.996 deg
};
P[211]{
   GP1:
    UF : 0, UT : 6,      CONFIG : 'N U T, 0, 0, 0',
    X =  321.148  mm,    Y =   11.557  mm,    Z =   -299.383  mm,
    W =  -183.835 deg,    P =   0.067 deg,    R =   -0.996 deg
};
P[212]{
   GP1:
    UF : 0, UT : 6,      CONFIG : 'N U T, 0, 0, 0',
    X =  321.105  mm,    Y =   16.605  mm,    Z =   -298.397  mm,
    W =  -183.603 deg,    P =   0.063 deg,    R =   -0.996 deg
};
P[213]{
   GP1:
    UF : 0, UT : 6,      CONFIG : 'N U T, 0, 0, 0',
    X =  321.235  mm,    Y =   22.058  mm,    Z =   -297.386  mm,
    W =  -183.292 deg,    P =   0.057 deg,    R =   -0.996 deg
};
P[214]{
   GP1:
    UF : 0, UT : 6,      CONFIG : 'N U T, 0, 0, 0',
    X =  320.964  mm,    Y =   27.368  mm,    Z =   -297.168  mm,
    W =  -182.807 deg,    P =   0.049 deg,    R =   -0.997 deg
};
P[215]{
   GP1:
    UF : 0, UT : 6,      CONFIG : 'N U T, 0, 0, 0',
    X =  321.240  mm,    Y =   32.975  mm,    Z =   -297.168  mm,
    W =  -181.893 deg,    P =   0.033 deg,    R =   -0.997 deg
};
P[216]{
   GP1:
    UF : 0, UT : 6,      CONFIG : 'N U T, 0, 0, 0',
    X =  320.683  mm,    Y =   95.475  mm,    Z =   -325.827  mm,
    W =  -180.000 deg,    P =   0.000 deg,    R =   0.000 deg
};
P[217]{
   GP1:
    UF : 0, UT : 6,      CONFIG : 'N U T, 0, 0, 0',
    X =  294.244  mm,    Y =   95.475  mm,    Z =   -325.827  mm,
    W =  -180.000 deg,    P =   0.000 deg,    R =   0.000 deg
};
P[218]{
   GP1:
    UF : 0, UT : 6,      CONFIG : 'N U T, 0, 0, 0',
    X =  296.089  mm,    Y =   35.828  mm,    Z =   -300.748  mm,
    W =  -179.092 deg,    P =   -0.016 deg,    R =   -0.990 deg
};
P[219]{
   GP1:
    UF : 0, UT : 6,      CONFIG : 'N U T, 0, 0, 0',
    X =  296.374  mm,    Y =   31.930  mm,    Z =   -300.748  mm,
    W =  -180.734 deg,    P =   0.013 deg,    R =   -0.991 deg
};
P[220]{
   GP1:
    UF : 0, UT : 6,      CONFIG : 'N U T, 0, 0, 0',
    X =  296.347  mm,    Y =   28.227  mm,    Z =   -300.748  mm,
    W =  -182.046 deg,    P =   0.035 deg,    R =   -0.991 deg
};
P[221]{
   GP1:
    UF : 0, UT : 6,      CONFIG : 'N U T, 0, 0, 0',
    X =  296.003  mm,    Y =   23.360  mm,    Z =   -300.594  mm,
    W =  -182.638 deg,    P =   0.046 deg,    R =   -0.992 deg
};
P[222]{
   GP1:
    UF : 0, UT : 6,      CONFIG : 'N U T, 0, 0, 0',
    X =  296.244  mm,    Y =   17.915  mm,    Z =   -300.378  mm,
    W =  -183.243 deg,    P =   0.056 deg,    R =   -0.992 deg
};
P[223]{
   GP1:
    UF : 0, UT : 6,      CONFIG : 'N U T, 0, 0, 0',
    X =  296.171  mm,    Y =   12.550  mm,    Z =   -300.728  mm,
    W =  -183.376 deg,    P =   0.059 deg,    R =   -0.993 deg
};
P[224]{
   GP1:
    UF : 0, UT : 6,      CONFIG : 'N U T, 0, 0, 0',
    X =  295.862  mm,    Y =   7.527  mm,    Z =   -301.242  mm,
    W =  -183.511 deg,    P =   0.061 deg,    R =   -0.993 deg
};
P[225]{
   GP1:
    UF : 0, UT : 6,      CONFIG : 'N U T, 0, 0, 0',
    X =  296.230  mm,    Y =   1.731  mm,    Z =   -302.483  mm,
    W =  -183.646 deg,    P =   0.063 deg,    R =   -0.993 deg
};
P[226]{
   GP1:
    UF : 0, UT : 6,      CONFIG : 'N U T, 0, 0, 0',
    X =  295.889  mm,    Y =   -3.316  mm,    Z =   -303.704  mm,
    W =  -183.725 deg,    P =   0.065 deg,    R =   -0.993 deg
};
P[227]{
   GP1:
    UF : 0, UT : 6,      CONFIG : 'N U T, 0, 0, 0',
    X =  294.953  mm,    Y =   -9.466  mm,    Z =   -305.086  mm,
    W =  -183.940 deg,    P =   0.068 deg,    R =   -0.993 deg
};
P[228]{
   GP1:
    UF : 0, UT : 6,      CONFIG : 'N U T, 0, 0, 0',
    X =  294.245  mm,    Y =   -21.489  mm,    Z =   -305.061  mm,
    W =  -184.174 deg,    P =   0.072 deg,    R =   -0.992 deg
};
P[229]{
   GP1:
    UF : 0, UT : 6,      CONFIG : 'N U T, 0, 0, 0',
    X =  296.259  mm,    Y =   -34.753  mm,    Z =   -307.836  mm,
    W =  -184.626 deg,    P =   0.080 deg,    R =   -0.991 deg
};
P[230]{
   GP1:
    UF : 0, UT : 6,      CONFIG : 'N U T, 0, 0, 0',
    X =  292.278  mm,    Y =   -38.766  mm,    Z =   -308.585  mm,
    W =  -185.232 deg,    P =   0.091 deg,    R =   -0.990 deg
};
P[231]{
   GP1:
    UF : 0, UT : 6,      CONFIG : 'N U T, 0, 0, 0',
    X =  295.904  mm,    Y =   -39.613  mm,    Z =   -309.440  mm,
    W =  -185.200 deg,    P =   0.090 deg,    R =   -0.990 deg
};
P[232]{
   GP1:
    UF : 0, UT : 6,      CONFIG : 'N U T, 0, 0, 0',
    X =  295.897  mm,    Y =   -45.268  mm,    Z =   -308.550  mm,
    W =  -185.734 deg,    P =   0.099 deg,    R =   -0.989 deg
};
P[233]{
   GP1:
    UF : 0, UT : 6,      CONFIG : 'N U T, 0, 0, 0',
    X =  296.142  mm,    Y =   -48.786  mm,    Z =   -307.683  mm,
    W =  -186.170 deg,    P =   0.107 deg,    R =   -0.988 deg
};
P[234]{
   GP1:
    UF : 0, UT : 6,      CONFIG : 'N U T, 0, 0, 0',
    X =  295.679  mm,    Y =   -53.698  mm,    Z =   -307.351  mm,
    W =  -186.859 deg,    P =   0.119 deg,    R =   -0.987 deg
};
P[235]{
   GP1:
    UF : 0, UT : 6,      CONFIG : 'N U T, 0, 0, 0',
    X =  296.247  mm,    Y =   -57.974  mm,    Z =   -321.164  mm,
    W =  -187.367 deg,    P =   0.127 deg,    R =   -0.986 deg
};
P[236]{
   GP1:
    UF : 0, UT : 6,      CONFIG : 'N U T, 0, 0, 0',
    X =  292.717  mm,    Y =   -62.176  mm,    Z =   -321.164  mm,
    W =  -187.688 deg,    P =   0.133 deg,    R =   -0.984 deg
};
P[237]{
   GP1:
    UF : 0, UT : 6,      CONFIG : 'N U T, 0, 0, 0',
    X =  296.147  mm,    Y =   -62.840  mm,    Z =   -321.164  mm,
    W =  -188.142 deg,    P =   0.141 deg,    R =   -0.985 deg
};
P[238]{
   GP1:
    UF : 0, UT : 6,      CONFIG : 'N U T, 0, 0, 0',
    X =  295.021  mm,    Y =   -65.029  mm,    Z =   -321.164  mm,
    W =  -188.168 deg,    P =   0.141 deg,    R =   -0.984 deg
};
P[239]{
   GP1:
    UF : 0, UT : 6,      CONFIG : 'N U T, 0, 0, 0',
    X =  296.279  mm,    Y =   -65.087  mm,    Z =   -321.164  mm,
    W =  -188.322 deg,    P =   0.144 deg,    R =   -0.984 deg
};
P[240]{
   GP1:
    UF : 0, UT : 6,      CONFIG : 'N U T, 0, 0, 0',
    X =  294.244  mm,    Y =   -95.475  mm,    Z =   -325.827  mm,
    W =  -180.000 deg,    P =   0.000 deg,    R =   0.000 deg
};
P[241]{
   GP1:
    UF : 0, UT : 6,      CONFIG : 'N U T, 0, 0, 0',
    X =  267.805  mm,    Y =   -95.475  mm,    Z =   -325.827  mm,
    W =  -180.000 deg,    P =   0.000 deg,    R =   0.000 deg
};
P[242]{
   GP1:
    UF : 0, UT : 6,      CONFIG : 'N U T, 0, 0, 0',
    X =  265.923  mm,    Y =   -60.494  mm,    Z =   -323.330  mm,
    W =  -187.547 deg,    P =   0.129 deg,    R =   -0.970 deg
};
P[243]{
   GP1:
    UF : 0, UT : 6,      CONFIG : 'N U T, 0, 0, 0',
    X =  266.433  mm,    Y =   -57.996  mm,    Z =   -323.330  mm,
    W =  -187.375 deg,    P =   0.126 deg,    R =   -0.972 deg
};
P[244]{
   GP1:
    UF : 0, UT : 6,      CONFIG : 'N U T, 0, 0, 0',
    X =  266.004  mm,    Y =   -52.815  mm,    Z =   -323.330  mm,
    W =  -186.839 deg,    P =   0.117 deg,    R =   -0.973 deg
};
P[245]{
   GP1:
    UF : 0, UT : 6,      CONFIG : 'N U T, 0, 0, 0',
    X =  266.123  mm,    Y =   -48.447  mm,    Z =   -314.525  mm,
    W =  -186.497 deg,    P =   0.111 deg,    R =   -0.974 deg
};
P[246]{
   GP1:
    UF : 0, UT : 6,      CONFIG : 'N U T, 0, 0, 0',
    X =  266.013  mm,    Y =   -43.526  mm,    Z =   -313.587  mm,
    W =  -185.920 deg,    P =   0.101 deg,    R =   -0.975 deg
};
P[247]{
   GP1:
    UF : 0, UT : 6,      CONFIG : 'N U T, 0, 0, 0',
    X =  265.647  mm,    Y =   -37.082  mm,    Z =   -313.612  mm,
    W =  -185.283 deg,    P =   0.090 deg,    R =   -0.976 deg
};
P[248]{
   GP1:
    UF : 0, UT : 6,      CONFIG : 'N U T, 0, 0, 0',
    X =  266.195  mm,    Y =   -31.772  mm,    Z =   -312.956  mm,
    W =  -184.790 deg,    P =   0.082 deg,    R =   -0.977 deg
};
P[249]{
   GP1:
    UF : 0, UT : 6,      CONFIG : 'N U T, 0, 0, 0',
    X =  266.313  mm,    Y =   -27.268  mm,    Z =   -312.538  mm,
    W =  -184.653 deg,    P =   0.080 deg,    R =   -0.977 deg
};
P[250]{
   GP1:
    UF : 0, UT : 6,      CONFIG : 'N U T, 0, 0, 0',
    X =  266.509  mm,    Y =   -23.839  mm,    Z =   -312.540  mm,
    W =  -184.576 deg,    P =   0.078 deg,    R =   -0.977 deg
};
P[251]{
   GP1:
    UF : 0, UT : 6,      CONFIG : 'N U T, 0, 0, 0',
    X =  266.264  mm,    Y =   -20.895  mm,    Z =   -312.391  mm,
    W =  -184.336 deg,    P =   0.074 deg,    R =   -0.978 deg
};
P[252]{
   GP1:
    UF : 0, UT : 6,      CONFIG : 'N U T, 0, 0, 0',
    X =  266.312  mm,    Y =   -13.332  mm,    Z =   -312.088  mm,
    W =  -184.026 deg,    P =   0.069 deg,    R =   -0.977 deg
};
P[253]{
   GP1:
    UF : 0, UT : 6,      CONFIG : 'N U T, 0, 0, 0',
    X =  265.732  mm,    Y =   -9.430  mm,    Z =   -311.863  mm,
    W =  -183.904 deg,    P =   0.067 deg,    R =   -0.976 deg
};
P[254]{
   GP1:
    UF : 0, UT : 6,      CONFIG : 'N U T, 0, 0, 0',
    X =  266.001  mm,    Y =   -4.242  mm,    Z =   -311.660  mm,
    W =  -183.601 deg,    P =   0.061 deg,    R =   -0.976 deg
};
P[255]{
   GP1:
    UF : 0, UT : 6,      CONFIG : 'N U T, 0, 0, 0',
    X =  266.901  mm,    Y =   0.525  mm,    Z =   -311.195  mm,
    W =  -183.430 deg,    P =   0.059 deg,    R =   -0.977 deg
};
P[256]{
   GP1:
    UF : 0, UT : 6,      CONFIG : 'N U T, 0, 0, 0',
    X =  266.305  mm,    Y =   6.359  mm,    Z =   -311.270  mm,
    W =  -183.158 deg,    P =   0.054 deg,    R =   -0.976 deg
};
P[257]{
   GP1:
    UF : 0, UT : 6,      CONFIG : 'N U T, 0, 0, 0',
    X =  266.393  mm,    Y =   11.454  mm,    Z =   -311.381  mm,
    W =  -182.603 deg,    P =   0.044 deg,    R =   -0.976 deg
};
P[258]{
   GP1:
    UF : 0, UT : 6,      CONFIG : 'N U T, 0, 0, 0',
    X =  266.340  mm,    Y =   17.771  mm,    Z =   -311.746  mm,
    W =  -182.025 deg,    P =   0.034 deg,    R =   -0.974 deg
};
P[259]{
   GP1:
    UF : 0, UT : 6,      CONFIG : 'N U T, 0, 0, 0',
    X =  265.708  mm,    Y =   25.844  mm,    Z =   -313.830  mm,
    W =  -181.289 deg,    P =   0.022 deg,    R =   -0.973 deg
};
P[260]{
   GP1:
    UF : 0, UT : 6,      CONFIG : 'N U T, 0, 0, 0',
    X =  266.891  mm,    Y =   29.965  mm,    Z =   -314.625  mm,
    W =  -180.828 deg,    P =   0.014 deg,    R =   -0.973 deg
};
P[261]{
   GP1:
    UF : 0, UT : 6,      CONFIG : 'N U T, 0, 0, 0',
    X =  266.301  mm,    Y =   35.615  mm,    Z =   -317.925  mm,
    W =  -180.218 deg,    P =   0.004 deg,    R =   -0.972 deg
};
P[262]{
   GP1:
    UF : 0, UT : 6,      CONFIG : 'N U T, 0, 0, 0',
    X =  266.372  mm,    Y =   40.358  mm,    Z =   -324.399  mm,
    W =  -179.642 deg,    P =   -0.006 deg,    R =   -0.972 deg
};
P[263]{
   GP1:
    UF : 0, UT : 6,      CONFIG : 'N U T, 0, 0, 0',
    X =  269.252  mm,    Y =   45.294  mm,    Z =   -324.399  mm,
    W =  -179.032 deg,    P =   -0.016 deg,    R =   -0.973 deg
};
P[264]{
   GP1:
    UF : 0, UT : 6,      CONFIG : 'N U T, 0, 0, 0',
    X =  266.492  mm,    Y =   47.581  mm,    Z =   -324.399  mm,
    W =  -178.862 deg,    P =   -0.019 deg,    R =   -0.970 deg
};
P[265]{
   GP1:
    UF : 0, UT : 6,      CONFIG : 'N U T, 0, 0, 0',
    X =  267.805  mm,    Y =   95.475  mm,    Z =   -325.827  mm,
    W =  -180.000 deg,    P =   0.000 deg,    R =   0.000 deg
};
P[266]{
   GP1:
    UF : 0, UT : 6,      CONFIG : 'N U T, 0, 0, 0',
    X =  241.366  mm,    Y =   95.475  mm,    Z =   -325.827  mm,
    W =  -180.000 deg,    P =   0.000 deg,    R =   0.000 deg
};
P[267]{
   GP1:
    UF : 0, UT : 6,      CONFIG : 'N U T, 0, 0, 0',
    X =  241.366  mm,    Y =   20.224  mm,    Z =   -325.693  mm,
    W =  -181.275 deg,    P =   0.021 deg,    R =   -0.956 deg
};
P[268]{
   GP1:
    UF : 0, UT : 6,      CONFIG : 'N U T, 0, 0, 0',
    X =  241.530  mm,    Y =   16.959  mm,    Z =   -325.693  mm,
    W =  -181.548 deg,    P =   0.026 deg,    R =   -0.957 deg
};
P[269]{
   GP1:
    UF : 0, UT : 6,      CONFIG : 'N U T, 0, 0, 0',
    X =  241.457  mm,    Y =   13.132  mm,    Z =   -325.693  mm,
    W =  -181.897 deg,    P =   0.032 deg,    R =   -0.958 deg
};
P[270]{
   GP1:
    UF : 0, UT : 6,      CONFIG : 'N U T, 0, 0, 0',
    X =  241.620  mm,    Y =   7.218  mm,    Z =   -324.907  mm,
    W =  -182.155 deg,    P =   0.036 deg,    R =   -0.959 deg
};
P[271]{
   GP1:
    UF : 0, UT : 6,      CONFIG : 'N U T, 0, 0, 0',
    X =  242.134  mm,    Y =   2.653  mm,    Z =   -325.296  mm,
    W =  -182.706 deg,    P =   0.045 deg,    R =   -0.960 deg
};
P[272]{
   GP1:
    UF : 0, UT : 6,      CONFIG : 'N U T, 0, 0, 0',
    X =  242.477  mm,    Y =   -7.513  mm,    Z =   -324.699  mm,
    W =  -183.049 deg,    P =   0.051 deg,    R =   -0.961 deg
};
P[273]{
   GP1:
    UF : 0, UT : 6,      CONFIG : 'N U T, 0, 0, 0',
    X =  243.196  mm,    Y =   -15.837  mm,    Z =   -324.708  mm,
    W =  -183.515 deg,    P =   0.059 deg,    R =   -0.963 deg
};
P[274]{
   GP1:
    UF : 0, UT : 6,      CONFIG : 'N U T, 0, 0, 0',
    X =  242.649  mm,    Y =   -38.248  mm,    Z =   -325.298  mm,
    W =  -185.056 deg,    P =   0.085 deg,    R =   -0.962 deg
};
P[275]{
   GP1:
    UF : 0, UT : 6,      CONFIG : 'N U T, 0, 0, 0',
    X =  241.366  mm,    Y =   -95.475  mm,    Z =   -325.827  mm,
    W =  -180.000 deg,    P =   0.000 deg,    R =   0.000 deg
};
P[276]{
   GP1:
    UF : 0, UT : 6,      CONFIG : 'N U T, 0, 0, 0',
    X =  400.000  mm,    Y =   0.000  mm,    Z =   -225.827  mm,
    W =  -180.000 deg,    P =   0.000 deg,    R =   0.000 deg
};
/END
